# B&R Automation Studio project Doctor
Automation Studio 4.9


## Configuration Doctoring

CPU 4PPC70.0702-20B, AutomationRuntime J4.93, Build 4.1.2, Safety 0.0, Vc V4.73.3

### Task classes (Cpu.sw)
```
Cyclic#1 (cycle 2000 us, tolerance 4000 us):
  HS_Inp_Doc <- Doctoring.HS_Inp_Doct.prg
  UnWindTC <- UnWindTC.prg [disabled]
Cyclic#4:
  HMI <- HMI.prg
  Alarms <- Alarms.prg
  EPLCom <- EPLCom.EPLCom.prg
DataObjects: Acp10sys
VcDataObjects: Vis <- Vis.dob
Binaries: udbdef, FWRules, TCData, vcctext, arialbd, vcpdi855, vcmgr, vcdsint, vcdsloc, vcbclass, vcfntttf, vctcal, vcshared, vcrt, vcpk, vccbmp, vcfile, vccbtn, vccslider, vccdt, vcptelo, vcalarm, vccnum, vcpdsw, arial, vccovl, vccalarm, vccstr, vcpdi815, vcpfppc7, vcgclass, vcpdihd, vcnet, Vis01, Vis03, vcpkat, Vis02, vcpdvnc, vccline, visvc, vclibvc, vcclbox, vccshape, acp10cfg, Acp10map, arconfig, User, iomap, asfw, ashwac, ashwd, sysconf, Role, vcpfar00, vcxml, vcchspot, vcchtml, vccurl, Vis_Re02, Vis_Re01, Vis_Re03, Vis_Re, vcctrend
Libraries: NcGlobal, sys_lib, brsystem, runtime, LoopConR, LoopCont, Acp10_MC, Acp10man, Acp10par, AsBrMath, Acp10sim, asstring, standard, vclib, visapi, AsEPL, astime, fileio, powerlnk, asieccon, dataobj, vcresman, Library
```

### Hardware
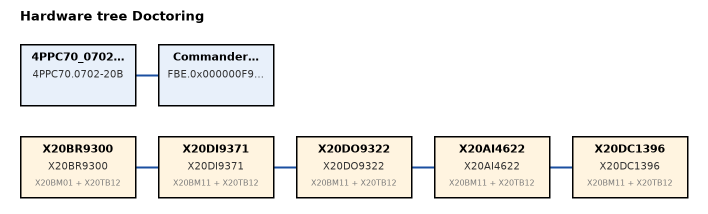
```
4PPC70_0702_20B : 4PPC70.0702-20B v1.5.4.0
  Connector IF1:
    CycleTime = 500
    MuxPrescaler = 2
  Connector IF2:
    ActivateDevice = 1
    Mode = Manual
    InternetAddress = 192.168.111.50
    SubnetMask = 255.255.255.0
    InaNodeNumber = 3
    Vnc1
    VncVcObjectName1 = Vis
    VncKeyMappingFile1 = VC\PS2-Keyboard.dis
    VncAuthentication1 = 1
    VncPasswordViewControl1 = v
    ActivateSnmp = 2
  Connector IF5:
    CycleTime = 1000
    BusLength = 500
  ConfigurationID = TensionCtl_Config1
  SimulationInaNodeNumber = 3
  PermanentPvSize = 5000
  RemanentGlobalPvSize = 10000
  EnableUsbRemoteInstall = 1
  EnableCfRemoteInstall = 1
  RebootReset = 2
  Connections = 8
  TimerDeviceType = EPLX2X
  TimerDevice = 4PPC70_0702_20B.IF1
  IdleTaskClass = 4
  TaskClassIdleTime = 4000
  Cyclic1Duration = 2000
  Cyclic1Tolerance = 4000
  Cyclic2Duration = 10000
  Cyclic5Duration = 500000
  Cyclic5Tolerance = 500000
  FileDevice1
  FileDeviceName1 = USER
  FileDevicePath1 = USER_PATH
  ActivateOpcUa = 1
  OpcUaInformationModels_PV_Version = 1
  VcObjectName = Vis
  KeyMappingFile = VC\4PPC70_0702_20B.dis
Commander_C200_OpenLoop : FBE.0x000000F9_Commander C200 OpenLoop vV01.01.12.04 (OrderNumber=Commander C200 OpenLoop)  [PLK1 -> 4PPC70_0702_20B.IF1 (NodeNumber=3) [Cable Type=PowerlinkCable, Length=10, Version=1.0.0.3]]
  Supervision = off
  DummyDeviceType = on
  p2001s05_direction = wo
  p2001s05_value = 5
  p2001s45_direction = ro
  p2004s01_direction = ro
  p2004s1A_direction = ro
  p2005s01_direction = ro
  p200As28_direction = ro
  p2014s15_value = 
X20AI4622 : X20AI4622 v1.5.0.0  [SS1 -> X20TB12g.SS; SL -> X20BM11f.SL1]
  Supervision = off
X20BM01 : X20BM01 v2.2.0.0
X20BM11b : X20BM11 v1.1.0.0  [X2X1 -> X20BM01.X2X2]
X20BM11d : X20BM11 v1.1.0.0  [X2X1 -> X20BM11b.X2X2]
X20BM11f : X20BM11 v1.1.0.0  [X2X1 -> X20BM11d.X2X2]
X20BM11h : X20BM11 v1.1.0.0  [X2X1 -> X20BM11f.X2X2]
X20BR9300 : X20BR9300 v1.3.0.0  [SS1 -> X20TB12.SS; SL -> X20BM01.SL1; X2X1 -> 4PPC70_0702_20B.IF5 [Cable Type=X2XCable, Length=10, Version=1.0.0.3]]
  Supervision = off
X20DC1396 : X20DC1396 v1.4.0.0  [SS1 -> X20TB12i.SS; SL -> X20BM11h.SL1]
  Supervision = off
X20DI9371 : X20DI9371 v1.6.0.0  [SS1 -> X20TB12c.SS; SL -> X20BM11b.SL1]
  Supervision = off
X20DO9322 : X20DO9322 v1.6.0.0  [SS1 -> X20TB12e.SS; SL -> X20BM11d.SL1]
  Supervision = off
  StatusInfo = off
X20TB12 : X20TB12 v1.0.0.0
X20TB12c : X20TB12 v1.0.0.0
X20TB12e : X20TB12 v1.0.0.0
X20TB12g : X20TB12 v1.0.0.0
X20TB12i : X20TB12 v1.0.0.0
```

### IoMap.iom - 4PPC70_0702_20B/IoMap.iom
```iecst
VAR_CONFIG
	::AI1[0] AT %IW."X20AI4622".AnalogInput01;
	::AI1[1] AT %IW."X20AI4622".AnalogInput02;
	::AI1[2] AT %IW."X20AI4622".AnalogInput03;
	::AI1[3] AT %IW."X20AI4622".AnalogInput04;
	::Enc_Value AT %IW."X20DC1396".Encoder01;
	::Data AT %IW."Commander_C200_OpenLoop".StatusWord_U16_I6041;
	::DataRead_INT AT %IW."Commander_C200_OpenLoop".Parameter40_StatusWord_I200A_S28;
	::DataTobeSent_UINT AT %QW."Commander_C200_OpenLoop".Parameter5_JogReference_I2001_S05Out;
	::DI1[0] AT %IX."X20DI9371".DigitalInput01;
	::DI1[1] AT %IX."X20DI9371".DigitalInput02;
	::DI1[2] AT %IX."X20DI9371".DigitalInput03;
	::DI1[3] AT %IX."X20DI9371".DigitalInput04;
	::DI1[4] AT %IX."X20DI9371".DigitalInput05;
	::DI1[5] AT %IX."X20DI9371".DigitalInput06;
	::DI1[6] AT %IX."X20DI9371".DigitalInput07;
	::DI1[7] AT %IX."X20DI9371".DigitalInput08;
	::DI1[8] AT %IX."X20DI9371".DigitalInput09;
	::DI1[9] AT %IX."X20DI9371".DigitalInput10;
	::DI1[10] AT %IX."X20DI9371".DigitalInput11;
	::DI1[11] AT %IX."X20DI9371".DigitalInput12;
	::DO1[0] AT %QX."X20DO9322".DigitalOutput01;
	::DO1[1] AT %QX."X20DO9322".DigitalOutput02;
	::DO1[2] AT %QX."X20DO9322".DigitalOutput03;
	::DO1[3] AT %QX."X20DO9322".DigitalOutput04;
	::DO1[4] AT %QX."X20DO9322".DigitalOutput05;
	::DO1[5] AT %QX."X20DO9322".DigitalOutput06;
	::DO1[6] AT %QX."X20DO9322".DigitalOutput07;
	::DO1[7] AT %QX."X20DO9322".DigitalOutput08;
	::DO1[8] AT %QX."X20DO9322".DigitalOutput09;
	::DO1[9] AT %QX."X20DO9322".DigitalOutput10;
	::DO1[10] AT %QX."X20DO9322".DigitalOutput11;
	::DO1[11] AT %QX."X20DO9322".DigitalOutput12;
END_VAR
```

## Configuration WndCLTensCtrl

### Hardware
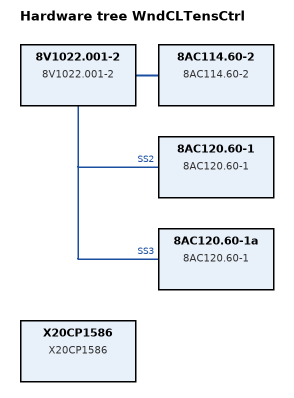
```
8AC114.60-2 : 8AC114.60-2 v1.0.0.8  [SS -> 8V1022.001-2.SS1; PLK1 -> X20CP1586.IF3 (NodeNumber=1) [Cable Type=PowerlinkCable, Length=10, Version=1.0.0.3]]
8AC120.60-1 : 8AC120.60-1 v2.2.0.0  [SS -> 8V1022.001-2.SS2]
8AC120.60-1a : 8AC120.60-1 v2.2.0.0  [SS -> 8V1022.001-2.SS3]
8V1022.001-2 : 8V1022.001-2 v2.2.0.0
  Simulate = complete
  ActiveMotorSimulation_r1 = on
  BothEndSwitchesAreNormallyOpen_r1 = on
  QuickStopIsNormallyOpen_r1 = on
X20CP1586 : X20CP1586 v1.10.0.0
  Connector IF1:
    ActivateIna = 0
  Connector IF2:
    ActivateDevice = 1
    EthInterfaceRedundant = 0
    InaPort = 11160
    Vnc1
    VncVcObjectName1 = Visu
    VncKeyMappingFile1 = VC\PS2-Keyboard.dis
    VncAuthentication1 = 1
    VncPasswordViewOnly1 = v
    VncPasswordViewControl1 = c
  Connector IF3:
    DNAConfiguration = manual
  ConfigurationID = TensionControl_Simulation
  Simulation = 1
  TimerDeviceType = SWIOTIMER
  SystemTick = 400
  TaskClassIdleTime = 400
  Cyclic1Duration = 400
  Cyclic1Tolerance = 0
  Cyclic2Duration = 800
  Cyclic2Tolerance = 0
  Cyclic3Duration = 10000
  Cyclic3Tolerance = 0
  Cyclic4Duration = 100000
  Cyclic4Tolerance = 100000
  Cyclic5Duration = 200000
  Cyclic5Tolerance = 200000
  Cyclic6Duration = 500000
  Cyclic6Tolerance = 500000
  Cyclic7Duration = 1000000
  Cyclic7Tolerance = 1000000
  Cyclic8Duration = 10000
  Cyclic8Tolerance = 30000000
```

## Logical view

Binary libraries used (declarations not repeated): Acp10sim 3.13.1, LoopCont 3.10.0

### Global.typ
```iecst
TYPE
	ActVal_typ : 	STRUCT
		Input_Val : INT;
		Output_Val : INT;
		Scale : Scale_typ;
	END_STRUCT;
	Act_para : 	STRUCT
		UnWindMPM : INT;
		UnWindTension : INT;
		UnWindRPM : INT;
		UnWindDia : INT;
		WindMPM : INT;
		WindTension : INT;
		WindRPM : INT;
		WindDia : INT;
		MainMPM : INT;
		MainRPM : INT;
		MainDia : USINT;
		InfeedTension : INT;
		OutfeedTension : INT;
		InfeedRPM : INT;
		OutfeedRPM : INT;
		InfeedMPM : INT;
		OutfeedMPM : INT;
	END_STRUCT;
	Ax_NonTensionCtl1 : 	STRUCT
		MPM : MPM_typ;
		Enable : BOOL;
		RPM : RPM_typ;
		Dia : Diameter_Scale;
		Drive : Drive_typ;
	END_STRUCT;
	Ax_TensionCtl : 	STRUCT
		Tension : Tension_typ;
		MPM : MPM_typ;
		Enable : BOOL;
		RPM : RPM_typ;
		Drive : Drive_typ;
		Dia : Diameter_Scale;
	END_STRUCT;
	Diameter_Scale : 	STRUCT
		InpMPM : INT;
		InpRPM : INT;
		ActDia : INT;
		MinDia : INT;
		MaxDia : INT;
	END_STRUCT;
	Drive_typ : 	STRUCT
		Freq_Scal : Scale_typ;
		RPM_Scal : Scale_typ;
		Trq_Scal : Scale_typ;
		Current_Scal : Scale_typ;
		ActFreq : INT;
		Status : USINT;
		ActualTrq : INT;
		ActualAmp : INT;
		ActRPM : INT;
		Fault : USINT;
	END_STRUCT;
	MPM_Scale : 	STRUCT
		InpDia : INT;
		InpRPM : INT;
		ActMPM : INT;
	END_STRUCT;
	MPM_typ : 	STRUCT
		SetMPM : INT;
		ActualMPM : INT;
		Enable : BOOL;
		Set : SetVal_typ;
		Actual : ActVal_typ;
	END_STRUCT;
	PIDPara_typ : 	STRUCT
		Y_max : INT;
		Y_min : INT;
		dY_max : REAL;
		Kp_sta : REAL;
		Tn_sta : REAL;
		Tv_sta : REAL;
		Tf_sta : REAL;
		WindDamp : REAL;
		Fbk_mode : REAL;
		d_mode : USINT;
		calc_mode : USINT;
		Attenu_val : REAL;
		Update : BOOL;
		Kp_mov : USINT;
		Tn_mov : USINT;
		Tv_mov : USINT;
		Tf_mov : USINT;
	END_STRUCT;
	RPM_Scale : 	STRUCT
		InpMPM : INT;
		InpDia : INT;
		ActRPM : INT;
		InpBits : INT;
	END_STRUCT;
	RPM_typ : 	STRUCT
		SetRPM : INT;
		ActualRPM : INT;
		Enable : BOOL;
		Set : SetVal_typ;
		Actual : ActVal_typ;
		PulsesPerRev : INT;
	END_STRUCT;
	Scale_typ : 	STRUCT
		InMin : INT;
		InMax : INT;
		OutMin : INT;
		OutMax : INT;
		Filter_tim : INT;
	END_STRUCT;
	SetVal_typ : 	STRUCT
		Output_Val : INT;
		Input_Val : INT;
		Scale : Scale_typ;
	END_STRUCT;
	Set_para : 	STRUCT
		MaxUnWindDia : INT;
		MaxWindDia : INT;
		MaxTorque : INT;
		MinUnWindDia : INT;
		MaxRPM : INT;
		MinRPM : INT;
		MinWindDia : INT;
		MinTorque : INT;
		MaxCurrent : INT;
		MinCurrent : INT;
		MainRoleDia : INT;
		MainMPM : INT;
		UnWindTension : INT;
		WindTension : INT;
		InfeedRolerDia : INT;
		OutfeedRolerDia : INT;
	END_STRUCT;
	Tension_Scale : 	STRUCT
		InpDia : INT;
		InpMPM : INT;
		ActTension : INT;
	END_STRUCT;
	Tension_typ : 	STRUCT
		Actual : ActVal_typ;
		Set : SetVal_typ;
		Enable : BOOL;
		SetTension : INT;
		ActualTension : INT;
	END_STRUCT;
	Ax_GeneralRef : 	STRUCT
		MPM : MPM_Scale;
		RPM : RPM_Scale;
		PulsesPerRev : INT;
	END_STRUCT;
END_TYPE
```

### Global.var
```iecst
VAR
	Actual : Act_para;
	AI1 : ARRAY[0..4] OF INT;
	AI2 : ARRAY[0..3] OF INT;
	AI3 : ARRAY[0..4] OF INT;
	Alarms : ARRAY[0..99] OF BOOL;
	Alarm_cnt : USINT;
	Alarm_new : BOOL;
	AO1 : ARRAY[0..3] OF INT;
	AxisDia : ARRAY[0..4] OF Diameter_Scale;
END_VAR
VAR RETAIN
	AxisKN : ARRAY[0..4] OF Tension_Scale;
END_VAR
VAR
	AxisMPM : ARRAY[0..4] OF MPM_Scale;
END_VAR
VAR RETAIN
	AxisRPM : ARRAY[0..4] OF RPM_Scale;
END_VAR
VAR
	Axis_KN : ARRAY[0..4] OF LCScINT;
	Axis_RPM : ARRAY[0..4] OF LCScINT;
	Axis_RpmInpFilt : ARRAY[0..4] OF LCPT1;
	CurrPage : USINT;
	DataRead_INT : INT;
	DataRead_UINT : UINT;
	DataTobeRead_INT : INT;
	DataTobeSent_UINT : UINT;
	DI1 : ARRAY[0..11] OF BOOL;
	DI2 : ARRAY[0..11] OF BOOL;
	DO1 : ARRAY[0..11] OF BOOL;
	DO2 : ARRAY[0..11] OF BOOL;
	DOUT1 : BOOL;
	DrvComm : BOOL;
	Enc_Value : INT;
	error : UINT;
END_VAR
VAR RETAIN
	Idler : Ax_GeneralRef;
END_VAR
VAR CONSTANT
	INFEED : USINT := 1;
END_VAR
VAR
	InFeed : Ax_TensionCtl;
	LastPage : USINT;
	LoginSuccessful : BOOL;
END_VAR
VAR CONSTANT
	MAIN : USINT := 4;
END_VAR
VAR
	MainDrive : Ax_NonTensionCtl1;
END_VAR
VAR CONSTANT
	MAX_AXES : USINT := 5;
END_VAR
VAR
	NewPage : USINT;
	NewPageReq : BOOL;
END_VAR
VAR CONSTANT
	OUTFEED : USINT := 2;
END_VAR
VAR
	OutFeed : Ax_TensionCtl;
	PageCall : BOOL;
	ParamChange : BOOL;
	PrevPage : USINT;
END_VAR
VAR CONSTANT
	PulsesPerRev : INT := 0;
END_VAR
VAR
	PulsesPerSec : INT;
	Set : Set_para;
	Statusdp_alarm : UINT;
	Statusdp_blink : UINT;
	status_gettime : UINT;
END_VAR
VAR RETAIN
	UnWind : Ax_TensionCtl;
END_VAR
VAR CONSTANT
	UNWINDER : USINT := 0;
END_VAR
VAR
	UnWindpara : LCPIDpara;
	UserAccessLevel : USINT;
END_VAR
VAR RETAIN
	Wind : Ax_NonTensionCtl1;
END_VAR
VAR CONSTANT
	WINDER : USINT := 3;
END_VAR
```

### Program Logical/5Drive/HS_Inp (IEC)

#### HS_Inp_Init.st - Init code
```iecst
PROGRAM _INIT
	(* Insert code here *)
	initialize	:= 1;

	(*Input of Tension Sensor for 4 axes except main drive *)
	AI1[0]	:= 0;	(*Unwinder Loadcell *)
	AI1[1]	:= 0;	(* Infeed Loadcell *)
	AI1[2]	:= 0;	(* Outfeed Loadcell *)
	AI1[3]	:= 0;	(* Winder Load cell *)
	AI1[4]	:= 0;	(* Dummy Load cell for Main Drive *)

	AI2[0]	:= 0;
	AI2[1]	:= 0;
	AI2[2]	:= 0;
	AI2[3]	:= 0; (*This input is configured for MAIN RPM calculation *)

	(* Input for RPM measurement from drive AI for 4 axes except Winder RPM*)
	AI3[0]	:= 0;   (* Unwinder RPM *)
	AI3[1]	:= 0;	(* Infeed RPM *)
	AI3[2]	:= 0;	(* Outfeed RPM *)
	AI3[3]	:= 0;	(* Winder RPM *)
	AI3[4]	:= 0;	(*This input is configured from AI2[3] for MAIN RPM *)

	AO1[0]	:= 0;
	AO1[1]	:= 0;
	AO1[2]	:= 0;
	AO1[3]	:= 0;

	DI1[0]	:= 0;
	DI1[1]	:= 0;
	DI1[2]	:= 0;
	DI1[3]	:= 0;
	DI1[4]	:= 0;
	DI1[5]	:= 0;
	DI1[6]	:= 0;
	DI1[7]	:= 0;
	DI1[8]	:= 0;
	DI1[9]	:= 0;
	DI1[10]	:= 0;
	DI1[11]	:= 0;

	DI2[0]	:= 0;
	DI2[1]	:= 0;
	DI2[2]	:= 0;
	DI2[3]	:= 0;
	DI2[4]	:= 0;
	DI2[5]	:= 0;
	DI2[6]	:= 0;
	DI2[7]	:= 0;
	DI2[8]	:= 0;
	DI2[9]	:= 0;
	DI2[10]	:= 0;
	DI2[11]	:= 0;

	DO1[0]	:= 0;
	DO1[1]	:= 0;
	DO1[2]	:= 0;
	DO1[3]	:= 0;
	DO1[4]	:= 0;
	DO1[5]	:= 0;
	DO1[6]	:= 0;
	DO1[7]	:= 0;
	DO1[8]	:= 0;
	DO1[9]	:= 0;
	DO1[10]	:= 0;
	DO1[11]	:= 0;

	DO2[0]	:= 0;
	DO2[1]	:= 0;
	DO2[2]	:= 0;
	DO2[3]	:= 0;
	DO2[4]	:= 0;
	DO2[5]	:= 0;
	DO2[6]	:= 0;
	DO2[7]	:= 0;
	DO2[8]	:= 0;
	DO2[9]	:= 0;
	DO2[10]	:= 0;
	DO2[11]	:= 0;

	i	:= 0;

	FOR i := 0 TO (MAX_AXES - 1) DO
		IF (AxisRPM[i].Fact.FilterTime = 0)THEN
			AxisRPM[i].Fact.FilterTime	:= 15;
		END_IF

		Axis_RpmInpFilt[i].enable		:= TRUE;
		Axis_RpmInpFilt[i].t			:= AxisRPM[i].Fact.FilterTime;
		Axis_RpmInpFilt[i].yset   		:= 0;
		Axis_RpmInpFilt[i].basetime 	:= HSCounter.mscnt;
		Axis_RpmInpFilt[i].set    		:= FALSE;
	END_FOR;

	FOR i :=0 TO (MAX_AXES - 1)BY 1 DO
		IF (AxisKN[i].Fact.FilterTime = 0)THEN
			AxisKN[i].Fact.FilterTime	:= 15;
		END_IF

		Axis_KNInpFilt[i].enable		:= TRUE;
		Axis_KNInpFilt[i].t				:= AxisKN[i].Fact.FilterTime;
		Axis_KNInpFilt[i].yset   		:= 0;
		Axis_KNInpFilt[i].basetime 		:= HSCounter.mscnt;
		Axis_KNInpFilt[i].set    		:= FALSE;
	END_FOR;

	FOR i := 0 TO (MAX_AXES - 1) BY 1 DO
		AxisRPM[i].InpBits		:= 0;
		AxisRPM[i].ActRPM		:= 0;

		Axis_RPM[i].x	:= AxisRPM[i].InpBits;
		Axis_RPM[i]();

		AxisKN[i].InpBits		:=	0;
		AxisKN[i].ActTension	:= 0;

		Axis_KN[i].x	:= AxisKN[i].InpBits;
		Axis_KN[i]();
	END_FOR;

	(* UnWinder & Infeed calculation initialization *)
	(*	UnWindFilt.enable	:= 1;
	UnWindFilt.set   	:= 1;
	UnWindFilt.t		:= 0.1;
	UnWindFilt.y_set	:= 0.0;
	UnWindFilt.x 		:= 0.0;
	UnWindFilt();
	UnWindFilt.set   	:= 0;

	ActUnWindKN.x1		:= UnWindKN.MinBits;
	ActUnWindKN.x2		:= UnWindKN.MaxBits;
	ActUnWindKN.y1		:= UnWindKN.MinTension;
	ActUnWindKN.y2		:= UnWindKN.MaxTension;

	InfeedFilt.enable	:= 1;
	InfeedFilt.set   	:= 1;
	InfeedFilt.t		:= 0.1;
	InfeedFilt.y_set	:= 0.0;
	InfeedFilt.x 		:= 0.0;
	InfeedFilt();
	InfeedFilt.set   	:= 0;

	ActInfeedKN.x1		:= InfeedKN.MinBits;
	ActInfeedKN.x2		:= InfeedKN.MaxBits;
	ActInfeedKN.y1		:= InfeedKN.MinTension;
	ActInfeedKN.y2		:= InfeedKN.MaxTension;
*)

	(* Winder & Outfeed calculation initialization *)

(*	WindFilt.enable		:= 1;
	WindFilt.set   		:= 1;
	WindFilt.t			:= 0.1;
	WindFilt.y_set		:= 0.0;
	WindFilt.x 			:= 0.0;
	WindFilt();
	WindFilt.set   		:= 0;

	ActWindKN.x1		:= WinderKN.MinBits;
	ActWindKN.x2		:= WinderKN.MaxBits;
	ActWindKN.y1		:= WinderKN.MinTension;
	ActWindKN.y2		:= WinderKN.MaxTension;

	OutfeedFilt.enable	:= 1;
	OutfeedFilt.set   	:= 1;
	OutfeedFilt.t		:= 0.1;
	OutfeedFilt.y_set	:= 0.0;
	OutfeedFilt.x 		:= 0.0;
	OutfeedFilt();
	OutfeedFilt.set   	:= 0;

	ActOutfeedKN.x1		:= OutfeedKN.MinBits;
	ActOutfeedKN.x2		:= OutfeedKN.MaxBits;
	ActOutfeedKN.y1		:= OutfeedKN.MinTension;
	ActOutfeedKN.y2		:= OutfeedKN.MaxTension;
*)

END_PROGRAM
```

### Program Logical/Doctoring/HS_Inp_Doct (IEC)

#### HS_Inp_Cyclic.st
```iecst
PROGRAM _CYCLIC
	// Time base counter
	HSCounter();

	IF(initialize = 1)THEN
		// Initialize all filters

		UnwindFilt.x	:= 0;
		UnwindFilt();

		WindFilt.x		:= 0;
		WindFilt();

		IF(UnWind.RPM.PulsesPerRev = 0)THEN
			UnWind.RPM.PulsesPerRev := 1;
		END_IF

		IF(Wind.RPM.PulsesPerRev= 0)THEN
			Wind.RPM.PulsesPerRev := 1;
		END_IF

		initialize := 0;

		Time_1sec.IN	:= 1;
		Old_EncValue	:= Enc_Value;

	ELSE
		// CALCULATE RPM AND MPM OF IDLER AXIS

		IF(Time_1sec.Q = 1)THEN
			PulsesPerMin	:= (Enc_Value - Old_EncValue)*60;
			Time_1sec.IN	:= 0;
		ELSIF (Time_1sec.IN = 0)THEN
			Old_EncValue	:= Enc_Value;
			Time_1sec.IN	:= 1;
		END_IF

		Idler.RPM.ActRPM := UDINT_TO_INT(PulsesPerMin)/Idler.PulsesPerRev;
		Idler.MPM.ActMPM := (314 * Idler.MPM.InpDia * Idler.RPM.ActRPM)/1000; // Idler Roller MPM (in 0.01 MPM) -> which is the system MPM

		//Filter the Winder & UnWinder RPM values read from the Drive
		UnwindFilt.x	:= DINT_TO_INT(UnWind.Drive.ActRPM/10);
		UnwindFilt();
		UnWind.RPM.Actual.Input_Val	:= UnwindFilt.y;

		WindFilt.x		:= DINT_TO_INT(Wind.Drive.ActRPM/10);
		WindFilt();
		Wind.RPM.Actual.Input_Val	:= WindFilt.y;

		//Calculate the RPM of Winder & Unwinder after filtering of Drive RPM & Scaling the value
		UnWindRPM_Scal.x		:= UnWind.RPM.Actual.Input_Val;
		UnWindRPM_Scal();
		UnWind.RPM.ActualRPM	:= UnWindRPM_Scal.y;

		WindRPM_Scal.x			:= Wind.RPM.Actual.Input_Val;
		WindRPM_Scal();
		Wind.RPM.ActualRPM		:= WindRPM_Scal.y;

		// CALCULATE DIAMETER OF WINDER AND UNWINDER
		IF(UnWind.RPM.ActualRPM > 0)THEN
			Numerator			:= INT_TO_UDINT(Idler.MPM.ActMPM * 1000);
			Denominator			:= INT_TO_UDINT(UnWind.RPM.ActualRPM * 314);
			UnWind.Dia.ActDia	:= UDINT_TO_INT(Numerator/Denominator) - UnWind.Dia.MinDia; // Winder DIA UNIT 0.01
		END_IF

		IF(Wind.RPM.ActualRPM > 0)THEN
			Numerator			:= INT_TO_UDINT(Idler.MPM.ActMPM * 1000);
			Denominator			:= INT_TO_UDINT(Wind.RPM.ActualRPM * 314);
			Wind.Dia.ActDia		:= UDINT_TO_INT(Numerator/Denominator) + Wind.Dia.MinDia; // Winder DIA UNIT 0.01
		END_IF

		//Just assign
		UnWind.Drive.ActFreq	:= UnWind.Drive.ActFreq;
		UnWind.Drive.ActRPM		:= UnWind.Drive.ActRPM;
		UnWind.Drive.ActualAmp	:= UnWind.Drive.ActualAmp;
		UnWind.Drive.ActualTrq	:= UnWind.Drive.ActualTrq;

	END_IF

	Time_1sec();

END_PROGRAM
```

### Program Logical/EPLCom/EPLCom

#### Init.st
```iecst
PROGRAM _INIT
	(* Insert code here *)
	(* Get NMT Status *)
	SDORead1.enable	:= 0;
	SDORead1.datalen := 4; //Data length, 2 bytes for 16-bit parameter
	SDORead1.pDevice := ADR(PLC_INTF); //POWERLINK interface on MN (PLC) ‘IF1’
	SDORead1.pData := ADR(NMT_Stat); //Data to be read into here
	SDORead1.node := 3; //Node address is set to 3
	SDORead1.index := 16#1000; //Read CAN related parameters starting from 0x1000 - 0x1fff
	SDORead1.subindex := 0;

	SDORead2.enable		:= 0;
	SDORead2.datalen := 4; //Data length, 2 bytes for 16-bit parameter
	SDORead2.pDevice := ADR(PLC_INTF); //POWERLINK interface on MN (PLC) ‘IF1’
	SDORead2.pData := ADR(Obj_Ident); //Data to be read into here
	SDORead2.node := 3; //Node address is set to 3
	SDORead2.index := 16#1018; //Read CAN related parameters starting from 0x1000 - 0x1fff
	SDORead2.subindex := 2;  //Read the product code from the drive

	DataReceived	:= 25;
	cnt_enable		:= 0;
	SDO_rd			:= 0;

END_PROGRAM
```

### Variables.var
```iecst
VAR
	UnWindFilt : LCPT1;
	UnWindPID : LCPID;
END_VAR
```

- Big_Fonts.fninfo (not shown)

- header.fninfo (not shown)

- Html_SDM.fninfo (not shown)

- Input_Bold.fninfo (not shown)

- Input_Normal.fninfo (not shown)

- globalArea.layer (not shown)

- msgBox.layer (not shown)

- ActualMPM.trd (not shown)

- SetTension.trd (not shown)

- Trend_1.tre (not shown)

Listed in the project but not available here: Logical/5Drive/HS_Inp/HS_Inp_Cyclic.st, Logical/5Drive/HS_Inp/HS_Inp_Exit.st, Logical/5Drive/HS_Inp/Types.typ, Logical/5Drive/HS_Inp/Variables.var
